FUNCTION_BLOCK DigitalLight
VAR_INPUT
	input: BOOL;
	keyType : INT;		//	0: Tap | 1: Toggle
END_VAR
VAR_OUTPUT
	output : BOOL;
	
END_VAR
VAR
	rtOnOff: R_TRIG;
END_VAR


IF keyType = 0 THEN
	rtOnOff(CLK:= input, Q=> );
	IF rtOnOff.Q THEN
		output := NOT output;
	END_IF
ELSIF keyType = 1 THEN
	output		:=	input;
ELSE
	output		:=	FALSE;
END_IF

END_FUNCTION_BLOCK

(* stored: Version 1.1.0.1, ProductVersion 3.1.4024.13
   POU DigitalLight: Id {e7c05c2b-c9cc-4ab1-9c73-c648a673d424}, SpecialFunc None *)
